FUNCTION_BLOCK FeederTags EXTENDS TcoCore.TcoObject
VAR
    _components : FeederTags_Components(THIS^);

    _homeMode : FeederTags_HomeMode(THIS^, eRestoreMode.None);
    _autoMode : FeederTags_AutoMode(THIS^, eRestoreMode.None);

    _homeModeTask : TcoCore.TcoTask(THIS^);
    _autoModeTask : TcoCore.TcoTask(THIS^);
    _serviceModeTask : TcoCore.TcoTask(THIS^);

    _assemblyTask : TcoCore.TcoTask(THIS^);

    _processTraceability : ProcessDataManager(THIS^);

    //Simulation counter
    _counter : DINT;
END_VAR

//SImualtion
_counter := _counter + 1;

_components();
_processTraceability();

HomeMode();
AutoMode();
ServiceMode();

METHOD AssemblySequenc : BOOL
VAR_INPUT
END_VAR
//IF (_assemblyTask.Execute()) THEN
////    Messenger.Trace('Grundstellungsfahrt aktiv');
//    _assemblySequence.Run();
//    _assemblyTask.DoneWhen(_assemblySequence.CurrentStep.ID = 999);
//END_IF
END_METHOD

METHOD AutoMode : BOOL
VAR_INPUT
END_VAR
_autoModeTask.Enabled := _homeModeTask.Done;

IF (_autoModeTask.Execute()) THEN
    Messenger.Trace('Auto Modus aktiv');
    _serviceModeTask.Abort();
    _autoMode.Run();
END_IF
END_METHOD

PROPERTY Components : reference to FeederTags_Components
GET
Components ref= _components;
END_GET
END_PROPERTY

PROPERTY Counter : reference to dint
GET
Counter ref= _counter;
END_GET
END_PROPERTY

METHOD HomeMode : BOOL
VAR_INPUT
END_VAR
IF (_homeModeTask.Execute()) THEN
    Messenger.Trace('Grundstellungsfahrt aktiv');
    _autoModeTask.Restore();
    _serviceModeTask.Restore();
    _homeMode.Run();
    _homeModeTask.DoneWhen(_homemode.CurrentStep.ID = 999);

    IF _homeModeTask.Done THEN
        _homeMode.Restore();
    END_IF
END_IF
END_METHOD

PROPERTY ProcessTraceAbility : REFERENCE TO ProcessDataManager
GET
ProcessTraceAbility REF= _processTraceability;
END_GET
END_PROPERTY

PROPERTY ProductionData : Reference to FeederTag_ProductionData
GET
ProductionData REF= _processTraceability._data;
END_GET
END_PROPERTY

METHOD ServiceMode : BOOL
IF(_serviceModeTask.Execute()) THEN
	Messenger.Trace('Schritt-Modus aktiv');	
	_autoModeTask.Restore();
	_homeModeTask.Restore();
	_homeMode.Restore();
	_autoMode.Restore();
	_components.Service();
END_IF
END_METHOD

END_FUNCTION_BLOCK

(* stored: Version 1.1.0.1, ProductVersion 3.1.4024.9
   POU FeederTags: Id {ddef14d8-19f9-04f0-273b-af4df910efa7}, SpecialFunc None
   Method AssemblySequenc: Id {429f0cfc-7d7e-0890-277d-d261344bba20}
   Method AutoMode: Id {2b27a906-75ff-085b-3206-47a5751ba104}
   Property Components: Id {76e2992d-231c-0d58-312c-50433fdad69d}
   Get Get: Id {d3bedfad-d653-050e-3388-39170c79c79e}
   Property Counter: Id {0d65ffe9-9746-0daa-3691-8afe7d54e334}
   Get Get: Id {3c4e4cd9-2353-0bfd-1353-39c5656697e7}
   Method HomeMode: Id {b2d0e6f0-ff19-0214-1afd-562a87a316dd}
   Property ProcessTraceAbility: Id {00f7b12c-b2ca-086c-1a2e-a6922d7e59d1}
   Get Get: Id {be6ddacb-fcc8-0d1b-3923-02d4bb84cc63}
   Property ProductionData: Id {4fe3bf27-fe79-02bf-1432-19e0065307dc}
   Get Get: Id {bc07ca47-bc4a-0d16-11db-3c9b709ae84a}
   Method ServiceMode: Id {1933e158-d53e-06b7-2013-f1a463ded5cd} *)
